# EPICS autosave request: motorApp/Db/motor_positions.req
# FILE... motor_positions.req
$(P)$(M).DVAL
